// TIA Portal V20 export
FUNCTION_BLOCK "COMP_VAL_==_OR_FB"   // FB30380, LAD
TITLE = COMP_VAL_==_OR_FB
{ S7_Optimized_Access := 'TRUE' }
AUTHOR : SICAR
FAMILY : Miscellaneous
VERSION : 1.0
// Der Baustein vergleicht die Werte der Eingänge IN1...IN8 mit dem Wert des Eingangs COMPARE_VALUE und verodert diese Vergleiche. Ist mindestens einer der Werte von IN1...IN8 gleich mit COMPARE_VALUE, so wird der Wert von COMPARE_VALUE in den Output VALUE geschrieben. Andernfalls wird VALUE mit dem Wert 0 beschrieben.
// UseCase: Damit kann ein "Summensignal" gebildet werden, z.B. für Produktionsdaten "LimitValues", womit ein Button animiert werden kann (Button "ProdData", "Grenzwerte").
// The block compares the values of the inputs IN1 ... IN8 with the value of the input COMPARE_VALUE and OR-operation these comparisons. If at least one of the values of IN1 ... IN8 is equal with COMPARE_VALUE, the value of COMPARE_VALUE is written to output VALUE. Otherwise, VALUE is written with the value 0. 
// UseCase: With this, a "summary signal" can be formed, e.g. for production data "LimitValues", with which a button can be animated (Button "ProdData", "Limit Values").
// stored: AutoNumber false, MemoryReserve 100, SetENOAutomatically false
   VAR_INPUT
      COMPARE_VALUE { ExternalAccessible := 'False'; ExternalVisible := 'False'; ExternalWritable := 'False'} : DWord;
      IN1 { ExternalAccessible := 'False'; ExternalVisible := 'False'; ExternalWritable := 'False'} : DWord;
      IN2 { ExternalAccessible := 'False'; ExternalVisible := 'False'; ExternalWritable := 'False'} : DWord;
      IN3 { ExternalAccessible := 'False'; ExternalVisible := 'False'; ExternalWritable := 'False'} : DWord;
      IN4 { ExternalAccessible := 'False'; ExternalVisible := 'False'; ExternalWritable := 'False'} : DWord;
      IN5 { ExternalAccessible := 'False'; ExternalVisible := 'False'; ExternalWritable := 'False'} : DWord;
      IN6 { ExternalAccessible := 'False'; ExternalVisible := 'False'; ExternalWritable := 'False'} : DWord;
      IN7 { ExternalAccessible := 'False'; ExternalVisible := 'False'; ExternalWritable := 'False'} : DWord;
      IN8 { ExternalAccessible := 'False'; ExternalVisible := 'False'; ExternalWritable := 'False'} : DWord;
   END_VAR
   VAR_OUTPUT
      VALUE { ExternalAccessible := 'False'; ExternalVisible := 'False'; ExternalWritable := 'False'} : DWord;
   END_VAR
   VAR_TEMP
      Dummy : Bool;
   END_VAR
BEGIN

REGION Network 1: VALUE = 0 schreiben / set VALUE = 0
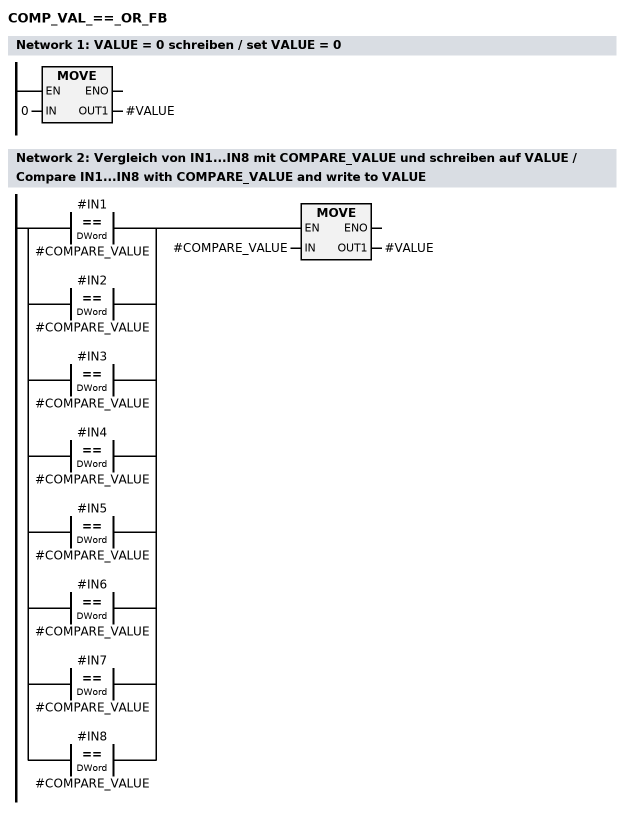
   RUNG wire#powerrail
      Move(in := 0, out1 => #VALUE)
   END_RUNG
   // the same network as SCL:
   #VALUE := 0;
END_REGION

REGION Network 2: Vergleich von IN1...IN8 mit COMPARE_VALUE und schreiben auf VALUE / Compare IN1...IN8 with COMPARE_VALUE and write to VALUE
   RUNG wire#powerrail
      { S7_Templates := "SrcType := DWord" } EQ_Contact(in1 := #IN1, in2 := #COMPARE_VALUE)
      wire#w1
      Move(in := #COMPARE_VALUE, out1 => #VALUE)
   END_RUNG
   RUNG wire#powerrail
      { S7_Templates := "SrcType := DWord" } EQ_Contact(in1 := #IN2, in2 := #COMPARE_VALUE)
   END_RUNG wire#w1
   RUNG wire#powerrail
      { S7_Templates := "SrcType := DWord" } EQ_Contact(in1 := #IN3, in2 := #COMPARE_VALUE)
   END_RUNG wire#w1
   RUNG wire#powerrail
      { S7_Templates := "SrcType := DWord" } EQ_Contact(in1 := #IN4, in2 := #COMPARE_VALUE)
   END_RUNG wire#w1
   RUNG wire#powerrail
      { S7_Templates := "SrcType := DWord" } EQ_Contact(in1 := #IN5, in2 := #COMPARE_VALUE)
   END_RUNG wire#w1
   RUNG wire#powerrail
      { S7_Templates := "SrcType := DWord" } EQ_Contact(in1 := #IN6, in2 := #COMPARE_VALUE)
   END_RUNG wire#w1
   RUNG wire#powerrail
      { S7_Templates := "SrcType := DWord" } EQ_Contact(in1 := #IN7, in2 := #COMPARE_VALUE)
   END_RUNG wire#w1
   RUNG wire#powerrail
      { S7_Templates := "SrcType := DWord" } EQ_Contact(in1 := #IN8, in2 := #COMPARE_VALUE)
   END_RUNG wire#w1
   // the same network as SCL:
   IF (#IN1 = #COMPARE_VALUE) OR (#IN2 = #COMPARE_VALUE) OR (#IN3 = #COMPARE_VALUE) OR (#IN4 = #COMPARE_VALUE) OR (#IN5 = #COMPARE_VALUE) OR (#IN6 = #COMPARE_VALUE) OR (#IN7 = #COMPARE_VALUE) OR (#IN8 = #COMPARE_VALUE) THEN
       #VALUE := #COMPARE_VALUE;
   END_IF;
END_REGION

NETWORK
TITLE = Baustein-Ende / End of block
// ENO immer "1" setzen mit SET & SAVE / ENO alwasy set "1" wtih SET & SAVE
      SET;
      SAVE;
END_FUNCTION_BLOCK
